INTERFACE I_ReceiverList EXTENDS Debug.I_Debug

METHOD Cap : UDINT
VAR_INPUT
END_VAR
END_METHOD

METHOD GetByPos : Results.Result
VAR_INPUT
	nPos			: UDINT;
END_VAR
VAR_OUTPUT
	iRec			: I_Receiver;
END_VAR
END_METHOD

METHOD GetByTag : Results.Result
VAR_INPUT
	iTag			: Tags.I_Tag;
END_VAR
VAR_OUTPUT
	iRec			: I_Receiver;
	nPos			: UDINT;
END_VAR
END_METHOD

METHOD GetExtender : ReceiverListExtender
VAR_INPUT
END_VAR
END_METHOD

METHOD IsReleased : BOOL
VAR_INPUT
END_VAR
END_METHOD

METHOD Length : UDINT
VAR_INPUT
END_VAR
END_METHOD

METHOD Release : ReceiverListExtender;
END_METHOD

END_INTERFACE

(* stored: Version 1.1.0.1
   Itf I_ReceiverList: Id {e8a2a3b3-d10e-4cf5-a30d-0a77b0b05371}
   Folder Get: Id {d92b47ff-ad9a-4196-87eb-590f6c09cd20}
   Folder Other: Id {af5639b7-e122-4cab-98d9-1e01a9c7319d}
   Method Cap: Id {b0c1213f-2e25-4c13-acac-070f696955ba}
   Method GetByPos: Id {efde4af8-f24c-4a23-93fd-995e70d10462}
   Method GetByTag: Id {2bd04f50-823d-4d69-bd00-b33edf082a6d}
   Method GetExtender: Id {b6650471-cd84-4a5e-916b-c4c1fd3c053a}
   Method IsReleased: Id {62ceecda-5d5c-4910-9fd1-312d81a9dacf}
   Method Length: Id {4030a647-51c5-4375-843b-67080467453e}
   Method Release: Id {9bf14676-deef-4d6f-b564-a92db3b2ee26} *)
